// TwinCAT 3 PLC project SerialComMaster
// ProgramVersion: 3.1.4026.12
// CompilerDefines: VISU_USEPROPERTYINFO
// libraries:
//   Tc2_ModbusRTU, * (Beckhoff Automation GmbH)
//   Tc2_SerialCom, * (Beckhoff Automation GmbH)
//   Tc2_Standard, * (Beckhoff Automation GmbH)
//   Tc2_System, * (Beckhoff Automation GmbH)
//   VisuSymbols, 4.5.0.0 (System)
// project tree:
//   / GlobalTextList.TcGTLO, PlcTask.TcTTO, Visualization Manager.TcVMO (not stored)
//   GVLs/ GVL_SerialCom.TcGVL
//   POUs/ MAIN.TcPOU, P_SerialCom.TcPOU
//   VISUs/ Visualization.TcVIS
// real-time tasks:
//   TASK PlcTask: cycle T#10ms, priority 20, ADS port 350

CONFIGURATION SerialComMaster
    RESOURCE PLC ON TwinCAT3
        TASK PlcTask(INTERVAL := T#10ms, PRIORITY := 20);
        PROGRAM MAIN WITH PlcTask : MAIN;
    END_RESOURCE
END_CONFIGURATION

// ---- GVLs/GVL_SerialCom.TcGVL
{attribute 'qualified_only'}
VAR_GLOBAL
	Inputs	:	ARRAY[0..255] OF WORD;		//入力レジスタModbusマスター読み取りのみ
	Outputs :	ARRAY[0..255] OF WORD;		//保持レジスタModbusマスター読み書き可能
	Memory 	:	ARRAY[0..255] OF WORD;		//Modbusマスター読み書き可能
END_VAR

// ---- POUs/MAIN.TcPOU
PROGRAM MAIN
VAR
END_VAR

P_SerialCom();

END_PROGRAM

// ---- POUs/P_SerialCom.TcPOU
PROGRAM P_SerialCom
VAR
	//テスト用のファンクションブロック
	fbSerialLineControlADS				:SerialLineControlADS;
	fbModbusRtuMasterV2_Generic			:ModbusRtuMasterV2_Generic;
	
	//テスト用の変数
	bConnect							:BOOL:=TRUE;
	stSerialCfg							:ComSerialConfig;
	RxBuffer							:ComBuffer;
	TxBuffer							:ComBuffer;
	bAdsError							:BOOL;
	nAdsErrorID							:UDINT;	
	
	bStart								:BOOL;

	i									:INT;

END_VAR

//---テスト用変数書き換え---
	i:=i+1;
	IF 32767 < i THEN
		i:=0;
	END_IF 
	
	GVL_SerialCom.Outputs[0]:=INT_TO_WORD(i);


//----テスト用のModbus通信---
	//シリアル接続を設定
	stSerialCfg.ComPort			:=3;
	stSerialCfg.Baudrate		:=19200;
	stSerialCfg.Parity			:=PARITY_EVEN;
	stSerialCfg.DataBits		:=8;
	stSerialCfg.StopBits		:=STOPBITS_ONE;
	stSerialCfg.DTR				:=DTR_CTRL_HANDSHAKE;
	stSerialCfg.RTS				:=RTS_CTRL_HANDSHAKE;
	stSerialCfg.CTS				:=FALSE;
	stSerialCfg.DSR				:=FALSE;
	
	//USB接続のシリアルポートで通信
	fbSerialLineControlADS(	Connect		:=bConnect,
							SerialCfg	:=stSerialCfg,
							NetId		:='192.168.15.16.1.1',
							Timeout		:=DEFAULT_ADS_TIMEOUT,
							TxBuffer	:=TxBuffer,
							RxBuffer	:=RxBuffer,
							PortOpened	=>,
							Error		=>bAdsError,
							ErrorID		=>nAdsErrorID,
							Busy		=>,
							TxBufCount	=>,
							RxBufCount	=>
							);
	
	//Modbus通信
	fbModbusRtuMasterV2_Generic.ReadWriteRegs(  UnitID				:=1,
												Quantity			:=120,
												MBAddr				:=16#0,
												cbLength			:=240,
												pMemoryAddr			:=ADR(GVL_SerialCom.Inputs),
												AuxQuantity			:=120,
												AuxMBAddr			:=16#800,
												AuxcbLength			:=240,
												pAuxMemoryAddr		:=ADR(GVL_SerialCom.Outputs),
												Execute				:=bStart,
												Timeout				:=DEFAULT_ADS_TIMEOUT,
												RxBuffer			:=RxBuffer,
												TxBuffer			:=TxBuffer,
												Busy				=>,
												Error				=>,
												ErrorId				=>,
												cbRead				=>
												);

END_PROGRAM

// ---- VISUs/Visualization.TcVIS
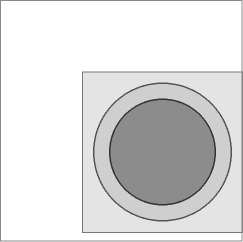
VISUALIZATION Visualization  // 243x242
    PushSwitch (82,62 161x180), variable: P_SerialCom.bStart, behaviour: TAP, style: Switch-PushSwitch-Gray
END_VISUALIZATION
